// TIA Portal V16 export
// export: Created 2023-03-29T11:03:45.2544791Z, ExportSetting WithDefaults, DisplayName Totally Integrated Automation Portal, DisplayVersion V16 Update 6, DisplayName TIA Portal Version Control Interface, DisplayVersion V16 Update 2, DisplayName TIA Portal Openness, DisplayVersion V16 Update 6, DisplayName STEP 7 Professional, DisplayVersion V16 Update 6, DisplayName STEP 7 Safety, DisplayVersion V16, DisplayName WinCC Advanced, DisplayVersion V16 Update 6
VAR_GLOBAL   // PLC tag table "Z8"
   inputAumagotowośćZ_8 AT %M69.0 : Bool;   // znacznik wejście
   setAlarm_Moment_Z_8 AT %M69.4 : Bool;   // znacznik alarmu od momentówki w trybie zdalnym (aut/mamnual)
   CMD_Awaria_Z_8 AT %M69.7 : Bool;   // Awaria zbiorcza
   isGotowość_Z_8 AT %M68.0 : Bool;   // bit gotowości wspólny
   inputAwariaMomentZ_8 AT %M68.5 : Bool;   // znacznik wejście
   inputOtwartaZ_8 AT %M68.2 : Bool;   // znacznik wejście
   Hbit_Reset_Z8 AT %M24.6 : Bool;
   setSVMO_Z_8 AT %M69.2 : Bool;   // Znacznik polecenia otwórz w trybie automat
   inputRuch_Z_8 AT %M68.4 : Bool;
   Hbit_Otwórz_Z8 AT %M24.4 : Bool;
   CMD_Close_Z_8 AT %M69.6 : Bool;   // załącz zamykanie
   inputAumaawariaZ_8 AT %M69.1 : Bool;   // znacznik wejście
   setSVMC_Z_8 AT %M69.3 : Bool;   // Znacznik polecenia zamknij w trybie automat
   Hbit_Alarm_Z8 AT %M24.0 : Bool;
   Hbit_Zamknij_Z8 AT %M24.5 : Bool;
   CMD_Open_Z_8 AT %M69.5 : Bool;   // załącz otwieranie
   inputZamkniętaZ_8 AT %M68.3 : Bool;   // znacznik wejście
   Hbit_Zamknieta_Z8 AT %M24.3 : Bool;
   inputREMT_Z_8 AT %M68.1 : Bool;   // znacznik wejście zdalne
   Hbit_REN_Z8 AT %M24.2 : Bool;
   isAUMA_Z_8 AT %M44.2 : Bool;   // przęłącznik wymiany na AUMA
   inputAumalokalneZ_8 AT %M68.6 : Bool;   // znacznik wejście
   Hbit_Otwarta_Z8 AT %M24.1 : Bool;
   Hbit_Auto_Manu_Z8 AT %M24.7 : Bool;
   Byte_Status_Z8 AT %MW24 : Word;   // Słowo statusu napędu
   inputAumaautomatZ_8 AT %M68.7 : Bool;   // znacznik wejście
   edge_Hz_Z8 AT %M92.3 : Bool;   // pamięć zbocza 1 Hz
END_VAR
